FUNCTION_BLOCK FB_GaugeLimit
VAR_INPUT
END_VAR
VAR_OUTPUT
END_VAR
VAR
END_VAR

END_FUNCTION_BLOCK

(* stored: Version 1.1.0.1, ProductVersion 3.1.4026.11
   POU FB_GaugeLimit: Id {e1309d19-0844-487d-9879-15c8a89df55d}, SpecialFunc None *)
